TYPE PARoute :
STRUCT
	_Items : ARRAY [1..GCL.cRouteItemMAX] OF IACEdge;	
	_IsResolved : BOOL;
	_IsAssigned : BOOL;
END_STRUCT
END_TYPE

(* stored: Version 1.1.0.1, ProductVersion 3.1.4020.12
   DUT PARoute: Id {c92aa8cc-5555-44b1-8330-1d1da5d2780c} *)
